TYPE udt_AdsAddr_AX5805 :
STRUCT
(*Used to read in the ADS address of the AX5805*)
(*Data structure must remain in this order*)
	Addr:		udt_AdsAddr;
	port:			UINT;
END_STRUCT
END_TYPE

(* stored: Version 1.1.0.1, ProductVersion 3.1.4024.9
   DUT udt_AdsAddr_AX5805: Id {6efd8bea-ea77-409c-af9d-e491d4f955eb} *)
